FUNCTION_BLOCK EnumeratorConnectionItem IMPLEMENTS I_EnumeratorConnectionItem
VAR
	enumeratorConnection : I_EnumeratorConnection;
END_VAR

METHOD FB_init : BOOL
VAR_INPUT
	bInitRetains : BOOL; // if TRUE, the retain variables are initialized (warm start / cold start)
	bInCopyCode : BOOL;  // if TRUE, the instance afterwards gets moved into the copy code (online change)
	EnumeratorConnection : I_EnumeratorConnection;
END_VAR
this^.enumeratorConnection := EnumeratorConnection;
END_METHOD

PROPERTY PUBLIC Get : I_EnumeratorConnection
GET
Get := enumeratorConnection;
END_GET
END_PROPERTY

END_FUNCTION_BLOCK

(* stored: Version 1.1.0.1, ProductVersion 3.1.4024.12
   POU EnumeratorConnectionItem: Id {04294803-447a-4de9-9c4c-db99f387c92c}, SpecialFunc None
   Folder Constructor: Id {b199530d-e76c-4723-80fd-0ce2e538e903}
   Method FB_init: Id {66df9481-f8bf-47c1-841c-452f16001c81}
   Property Get: Id {c3f57684-bb31-43ea-a067-8c18357cca34}
   Get Get: Id {78655108-915f-47d5-8c54-e9f30c102d41} *)
